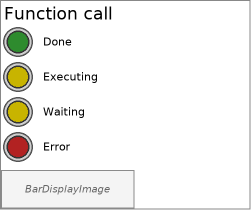
VISUALIZATION _VisuFunctionCall  // 251x210
    Label (1,1 248x25), "Function call"
    Lamp1 (1,25 34x34), variable: ComGVL._fbTryOutDone, style: Lamp-Lamp1-Green
    Lamp1 (1,60 34x34), variable: ComGVL._fbTryOutExecuting, style: Lamp-Lamp1-Yellow
    Lamp1 (1,95 34x34), variable: ComGVL._fbTryOutWaiting, style: Lamp-Lamp1-Yellow
    Lamp1 (1,130 34x34), variable: ComGVL._fbTryOutError, style: Lamp-Lamp1-Red
    BarDisplayImage (1,170 133x38), value: ComGVL._fbTryOutProgress, style: BarDisplayImage-Gray, scale format: %.1f, scale 0..100
    Label (40,25 100x34), "Done"
    Label (40,60 100x34), "Executing"
    Label (40,95 100x34), "Waiting"
    Label (40,130 100x34), "Error"
END_VISUALIZATION

(* stored: Version 1.1.0.1, ProductVersion 3.1.4024.2
   Visu _VisuFunctionCall: Id {3ab90189-9257-4e63-b7a6-8769999a2097} *)
